FUNCTION_BLOCK ST_REC_CONN (* Reconnects an event or data connection between two FB instances *)
  (* Standard: 61499-1; Classification: Reconfiguration; Function: Reconnects Connection; Type: Structural Service; Description: Copyright (c) 2012 Profactor GmbH This program and the accompanying materials are made available under the terms of the Eclipse Public License 2.0 which is available at https://www.eclipse.org/legal/epl-2.0/ SPDX-License-Identifier: EPL-2.0 *)
  (* Version 1.0, 2012-05-31, Gerhard Ebenhofer, Profactor GmbH *)
  (* Compiler Cpp GNU GCC >3.0 *)
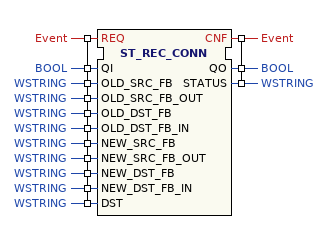
  EVENT_INPUT
    REQ WITH OLD_SRC_FB, OLD_SRC_FB_OUT, OLD_DST_FB, OLD_DST_FB_IN, DST, NEW_SRC_FB, NEW_SRC_FB_OUT, NEW_DST_FB, NEW_DST_FB_IN, QI; (* Event to require reconnection of a connection *)
  END_EVENT
  EVENT_OUTPUT
    CNF WITH STATUS, QO; (* Event to confirm that the reconnection of the connection has been carried out *)
  END_EVENT
  VAR_INPUT
    QI : BOOL; (* Event Input Qualifier *)
    OLD_SRC_FB : WSTRING; (* Reference to old Source FB instance *)
    OLD_SRC_FB_OUT : WSTRING; (* Reference to old Source FB instance Event/Data-Output *)
    OLD_DST_FB : WSTRING; (* Reference to old Destination FB instance *)
    OLD_DST_FB_IN : WSTRING; (* Reference to old Destination FB instance Event/Data-Input *)
    NEW_SRC_FB : WSTRING; (* Reference to new Source FB instance *)
    NEW_SRC_FB_OUT : WSTRING; (* Reference to new Source FB instance Event/Data-Output *)
    NEW_DST_FB : WSTRING; (* Reference to new Destination FB instance *)
    NEW_DST_FB_IN : WSTRING; (* Reference to new Destination FB instance Event/Data-Input *)
    DST : WSTRING; (* Destination where the connection has to be reconnected (Syntax: ResourceName) *)
  END_VAR
  VAR_OUTPUT
    QO : BOOL; (* Event Output Qualifier *)
    STATUS : WSTRING; (* Service Status: RDY, NO_SUCH_OBJECT, INVALID_STATE *)
  END_VAR
END_FUNCTION_BLOCK
